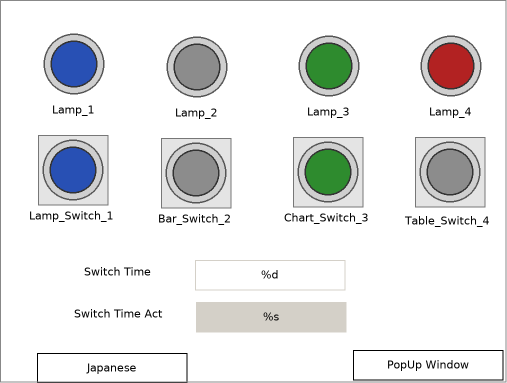
VISUALIZATION P01_Swtich_Lamp  // 507x383
    Lamp1 (39,29 70x70), variable: Main.bHmi_LAMP1, style: Lamp-Lamp1-Blue
    Label (17,95 113x30), "Lamp_1"
    PushSwitch (38,135 70x70), variable: Main.bHmi_Swtic1, behaviour: TOGGLE, style: Switch-PushSwitch-Blue
    Label (15,201 113x30), "Lamp_Switch_1"
    Lamp1 (162,32 70x70), variable: Main.bHmi_LAMP2, style: Lamp-Lamp1-Gray
    Label (140,98 113x30), "Lamp_2"
    PushSwitch (161,138 70x70), variable: Main.bHmi_Swtic2, behaviour: TOGGLE, style: Switch-PushSwitch-Gray
    Label (138,204 113x30), "Bar_Switch_2"
    Lamp1 (294,31 70x70), variable: Main.bHmi_LAMP3, style: Lamp-Lamp1-Green
    Label (272,97 113x30), "Lamp_3"
    PushSwitch (293,137 70x70), variable: Main.bHmi_Swtic3, behaviour: TOGGLE, style: Switch-PushSwitch-Green
    Label (270,203 113x30), "Chart_Switch_3"
    Lamp1 (416,31 70x70), variable: Main.bHmi_LAMP4, style: Lamp-Lamp1-Red
    Label (394,97 113x30), "Lamp_4"
    PushSwitch (415,137 70x70), variable: Main.bHmi_Swtic4, behaviour: TOGGLE, style: Switch-PushSwitch-Gray
    Label (391,206 113x30), "Table_Switch_4"
    Textfield (195,260 150x30), "%d", text variable: Main.iIN_VOLUME
        OnMouseUp: write the text variable via Default
    Label (61,257 113x30), "Switch Time"
    Textfield (196,302 150x30), "%s", text variable: MAIN.fbBlinker.T1.ET
    Label (62,299 113x30), "Switch Time Act"
    RoundedRectangle (37,353 150x30), "Japanese"
        OnMouseClick: ChangeLanguage ChangeLanguage=JP
    RoundedRectangle (353,350 150x30), "PopUp Window"
        OnMouseClick: OpenDialog Dialog=W01_PopupScreen, OpenModal=True, OpenCentered=True
END_VISUALIZATION

(* stored: Version 1.1.0.1, ProductVersion 3.1.4024.6
   Visu P01_Swtich_Lamp: Id {a528be18-4486-4717-a5d6-f8ac8d94750f} *)
